Staubli VAL3: Control_Point.pgx

public program Control_Point(pointRx& x_pP)
  local string l_sItem[6]
  local num l_nNum
  local num l_nKey
  local num l_nData[6]
  local num l_nSelectIndex
begin

  //修改点位的 joint
  l_nData[0]=x_pP.trsf.x
  l_nData[1]=x_pP.trsf.y
  l_nData[2]=x_pP.trsf.z
  l_nData[3]=x_pP.trsf.rx
  l_nData[4]=x_pP.trsf.ry
  l_nData[5]=x_pP.trsf.rz

  l_sItem[0]="X    :"+toString(".3",l_nData[0])
  l_sItem[1]="y    :"+toString(".3",l_nData[1])
  l_sItem[2]="Z    :"+toString(".3",l_nData[2])
  l_sItem[3]="RX   :"+toString(".3",l_nData[3])
  l_sItem[4]="RY   :"+toString(".3",l_nData[4])
  l_sItem[5]="RZ   :"+toString(".3",l_nData[5])

  call Control_BottomS(",,,,,,取消,确定")
  call Control_PanelXY(8,0,15,6)
  call Control_Panel("Point值")
  call Control_List(l_sItem,l_nSelectIndex)
  while true
    l_nKey=getKey()

    switch l_nKey
      case 261
        l_nSelectIndex=max(0,l_nSelectIndex-1)
      break

      case 266
        l_nSelectIndex=min(l_nSelectIndex+1,5)
      break

      case 278
        x_pP.trsf.x=l_nData[0]
        x_pP.trsf.y=l_nData[1]
        x_pP.trsf.z=l_nData[2]
        x_pP.trsf.rx=l_nData[3]
        x_pP.trsf.ry=l_nData[4]
        x_pP.trsf.rz=l_nData[5]
         cls()
        return
      break


      case 277,255

        cls()
        return
      break

      case 270
        call Float_Edit(l_nData[l_nSelectIndex],nPanelLTopX+7,l_nSelectIndex+nPanelLTopY+1)
      break

    endSwitch

    if l_nKey!=-1
      l_sItem[0]="X    :"+toString(".3",l_nData[0])
      l_sItem[1]="y    :"+toString(".3",l_nData[1])
      l_sItem[2]="Z    :"+toString(".3",l_nData[2])
      l_sItem[3]="RX   :"+toString(".3",l_nData[3])
      l_sItem[4]="RY   :"+toString(".3",l_nData[4])
      l_sItem[5]="RZ   :"+toString(".3",l_nData[5])
      call Control_List(l_sItem,l_nSelectIndex)

    endIf






  endWhile





end
